// Project Hardware Driver layer. This is the only POU that accesses GVL_PressIO.
// It maps raw process-image symbols to semantic HALs and refreshes the Core
// topology publisher. It contains no sequence, mode, recipe or device behavior.
FUNCTION_BLOCK FB_PressIoDriver
VAR_OUTPUT
    // Raw N54 D2 operator buttons, republished so MAIN can drive Control On/Off
    // from hardware without becoming a second GVL_PressIO consumer.
    ControlOnButton  : BOOL;
    ControlOffButton : BOOL;
END_VAR
VAR
    _publisher : FB_IoTopologyPublisher;
    {attribute 'OPC.UA.DA' := '0'}
    _unit : REFERENCE TO FB_PressDemoUnit;
    _attached : BOOL;
    // Hardware Control-On adapter: reconstructs the safety-status mirrors from
    // the raw relay/sensor process image on a machine with a hardwired N54 D2
    // Control On circuit (no TwinSAFE controller). Status only; not a safety fn.
    _controlOn : FB_PressControlOnCircuit;
    // Reads the REAL EtherCAT slave states from the master and publishes each
    // node's live state — the fieldbus tree reflects hardware, not Control-On.
    _busHealth : FB_EcBusHealth;
END_VAR

;

METHOD Setup : BOOL
VAR_INPUT
    UnitRef : REFERENCE TO FB_PressDemoUnit;
END_VAR
VAR
    // Left all-zero: FB_EcBusHealth auto-detects the EtherCAT master's AmsNetId,
    // so the project needs no fieldbus address and no XAE link. Assign a value
    // here only for a non-standard master (remote, or several on one PC).
    ecMasterNetId : T_AmsNetIdArr;
END_VAR
_unit REF= UnitRef;
_attached := _publisher.Setup(DataRef := GVL_PressFieldbus.Topology, ResetData := FALSE)
    AND __ISVALIDREF(_unit);
// Map the press topology to the EtherCAT master's slaves. The catalog defines
// node 1 = CX2030 master and nodes 2..6 = the five devices in the project tree
// (EK1200 coupler, EL1809, EL2809, EL6001, EL9011).
//
// Only THREE of those are slaves the master enumerates: the EK1200 coupler and
// the EL9011 end cap carry the bus but have no EtherCAT slave controller on the
// process-data ring, so they never appear in FB_EcGetAllSlaveStates. Declaring
// SlaveCount := 5 made the master's slave i land on catalog node i, shifting
// every state onto its neighbour: the EL6001's OP was published onto the
// EL2809, and the EL6001 itself read OFFLINE while it was perfectly healthy.
// State the mapping instead of assuming it.
_busHealth.Setup(Publisher := _publisher, MasterNetIdArr := ecMasterNetId,
    FirstSlaveNode := 3, SlaveCount := 3, MasterNodeIndex := 1);
_busHealth.M_MapSlaveNode(SlaveIndex := 1, NodeIndex := 3);   // EL1809
_busHealth.M_MapSlaveNode(SlaveIndex := 2, NodeIndex := 4);   // EL2809
_busHealth.M_MapSlaveNode(SlaveIndex := 3, NodeIndex := 5);   // EL6001
_busHealth.M_MapPassiveNode(NodeIndex := 2);                  // EK1200 coupler
_busHealth.M_MapPassiveNode(NodeIndex := 6);                  // EL9011 end cap
Setup := _attached;
END_METHOD

METHOD M_ReadInputs
VAR_IN_OUT
    PressHal : ST_CylinderHal;
    DoorHal : ST_CylinderHal;
    SlideHal : ST_CylinderHal;
    TwoHandHal : ST_TwoHandHal;
    PowerHal : ST_PowerGroupHal;
    PartPresentHal : ST_DigitalInputHal;
    AirPressureHal : ST_AirPressureHal;
    RawEStopHealthy : BOOL;
    SafeEStopOk : BOOL;
    SafeGuardClosed : BOOL;
    SafeTwoHandActive : BOOL;
    SafePneumaticPermit : BOOL;
    SafetyFieldbusHealthy : BOOL;
    StandardIoHealthy : BOOL;
END_VAR
VAR
    // EtherCAT process-image validity, DETECTED from the fieldbus master by the
    // library (FB_EcBusHealth) — the project no longer declares/links a RealBusOk.
    busOk : BOOL;
END_VAR
busOk := _busHealth.M_BusOk();
// Physical feeder retracted = logical slide inside; extended = outside.
SlideHal.ExtendedFb := GVL_PressIO._101B301A;
SlideHal.RetractedFb := GVL_PressIO._101B301B;
DoorHal.ExtendedFb := GVL_PressIO._101B201A;
DoorHal.RetractedFb := GVL_PressIO._101B201B;
PressHal.ExtendedFb := GVL_PressIO._101B202A;
PressHal.RetractedFb := GVL_PressIO._101B202B;
TwoHandHal.RightPressed := GVL_PressIO._101S101;
TwoHandHal.LeftPressed := GVL_PressIO._101S102;
PartPresentHal.Value := GVL_PressIO._101B601;
AirPressureHal.LowPressure := GVL_PressIO._000MB085A_2;
AirPressureHal.OperatingPressure := GVL_PressIO._000MB085A_4;
PowerHal.PowerFeedback := GVL_PressIO._000K911_Y32;
// This machine's safety is a hardwired N54 D2 Control On relay chain, not a
// TwinSAFE controller, so the GVL_PressSafety AT %I* aliases are never written.
// Reconstruct the read-only safety-status mirrors from the raw relay/sensor
// process image via the Control-On adapter. The relay chain remains the safety
// authority; these values drive HMI/interlock display only.
_controlOn.M_Evaluate(
    // POLARITY: =000+S1-K910A:14 is "Emergency Switch 1 PRESSED" (N54 D2), and on
    // THIS machine the contact is CONFIRMED NORMALLY OPEN - not pressed reads
    // FALSE, pressed reads TRUE - so inverting it yields the "healthy" mirror
    // this adapter publishes. Read un-inverted, a healthy machine reported
    // E-stop-unhealthy and control power was withheld (POWER_ENABLE_WITHHELD)
    // even with the relay chain demonstrably closed.
    //
    // DEMO WIRING ONLY - NOT FAIL-SAFE. A normally-open E-stop contact cannot
    // distinguish "not pressed" from a broken wire, a pulled terminal or a dead
    // input card: all read FALSE, and this mirror would then report HEALTHY.
    // ISO 13850 / EN 60204-1 require a normally-CLOSED contact so that any break
    // forces the stop. A production machine must rewire to NC and drop this
    // inversion. This mirror is diagnostic only - the hardwired relay chain
    // remains the safety authority (Core Sec.9), which is what keeps the
    // non-fail-safe wiring tolerable on a demo rig and nowhere else.
    EStopHealthyMirror := NOT GVL_PressIO._000K910A,
    DoorClosed := GVL_PressIO._101B201A,
    LeftButton := GVL_PressIO._101S102,
    RightButton := GVL_PressIO._101S101,
    ControlOnFeedback := GVL_PressIO._000K911_Y32,
    BusOk := busOk,
    ControlOnButton := GVL_PressIO._000BS901,
    ControlOffButton := GVL_PressIO._000BS902,
    AirPressureOk := GVL_PressIO._000MB085A_4 AND NOT GVL_PressIO._000MB085A_2);
RawEStopHealthy := _controlOn.RawEStopHealthy;
SafeEStopOk := _controlOn.SafeEStopOk;
SafeGuardClosed := _controlOn.SafeGuardClosed;
SafeTwoHandActive := _controlOn.SafeTwoHandActive;
SafePneumaticPermit := _controlOn.SafePneumaticPermit;
SafetyFieldbusHealthy := _controlOn.SafetyFieldbusHealthy;
StandardIoHealthy := _controlOn.StandardIoHealthy;
PartPresentHal.Quality := StandardIoHealthy;
AirPressureHal.Quality := StandardIoHealthy;
ControlOnButton := GVL_PressIO._000BS901;
ControlOffButton := GVL_PressIO._000BS902;
END_METHOD

// Also withdraws every held §10.5.1 force: under USE_SIMULATION no physical
// output is driven at all, so a set-point armed earlier must not survive here
// and reappear the moment a real write path runs (§10.5.1 rule 3).
METHOD M_ClearOutputs
_publisher.M_ApplyForces(Enabled := FALSE);
GVL_PressIO._101K301A := FALSE; GVL_PressIO._101K301B := FALSE;
GVL_PressIO._101K201A := FALSE; GVL_PressIO._101K201B := FALSE;
GVL_PressIO._101K202A := FALSE; GVL_PressIO._101K202B := FALSE;
GVL_PressIO._101P101 := FALSE; GVL_PressIO._101P102 := FALSE;
GVL_PressIO._000K951_A1 := FALSE; GVL_PressIO._000K911_A1 := FALSE;
END_METHOD

METHOD M_WriteOutputs
VAR_INPUT
    PressHal : ST_CylinderHal;
    DoorHal : ST_CylinderHal;
    SlideHal : ST_CylinderHal;
    PowerHal : ST_PowerGroupHal;
    LampsOn : BOOL;
    ControlCircuitMappingConfirmed : BOOL;
    // Core §10.5.1 rule 3 - FB_UnitBase.M_ForcePermitted() of the owning Unit.
    // The SAME predicate its ForceChannel accepted the request with, so a force
    // can never be accepted under conditions in which it would not be applied,
    // and leaving idle MANUAL withdraws every held set-point on that scan.
    ForcePermitted : BOOL;
END_VAR
// One call decides whether held set-points apply this scan, and withdraws them
// all on the falling edge. It runs BEFORE the writes below, so the very scan
// the Unit leaves idle MANUAL is already driven by application logic again.
_publisher.M_ApplyForces(Enabled := ForcePermitted);
// M_EffectiveBool returns the value, so each line still reads as the plain
// assignment it was: the application value, or the held force set-point while
// forcing is permitted and this channel is forced.
GVL_PressIO._101K301A := _publisher.M_EffectiveBool(NodeIndex := 4, ChannelIndex := 1, Value := SlideHal.ExtendOut);
GVL_PressIO._101K301B := _publisher.M_EffectiveBool(NodeIndex := 4, ChannelIndex := 2, Value := SlideHal.RetractOut);
GVL_PressIO._101K201A := _publisher.M_EffectiveBool(NodeIndex := 4, ChannelIndex := 3, Value := DoorHal.ExtendOut);
GVL_PressIO._101K201B := _publisher.M_EffectiveBool(NodeIndex := 4, ChannelIndex := 4, Value := DoorHal.RetractOut);
GVL_PressIO._101K202A := _publisher.M_EffectiveBool(NodeIndex := 4, ChannelIndex := 5, Value := PressHal.ExtendOut);
GVL_PressIO._101K202B := _publisher.M_EffectiveBool(NodeIndex := 4, ChannelIndex := 6, Value := PressHal.RetractOut);
GVL_PressIO._101P101 := _publisher.M_EffectiveBool(NodeIndex := 4, ChannelIndex := 7, Value := LampsOn);
GVL_PressIO._101P102 := _publisher.M_EffectiveBool(NodeIndex := 4, ChannelIndex := 8, Value := LampsOn);
// Ch9/Ch10 (_000K951_A1 / _000K911_A1) are never routed through the force
// path: they drive the hardwired N54 D2 Control On relay chain and the
// catalog never marks them forceable (§10.5.1 rule 4).
IF ControlCircuitMappingConfirmed THEN
    // N54 D2: these are DIFFERENT signals. SwitchControlOn is the momentary
    // button coil (2 s pulse); EnableControlOn is the bus/air permissive that
    // must be TRUE whenever the machine is healthy. Driving both from one power
    // request was why the control circuit could never energize.
    GVL_PressIO._000K951_A1 := _controlOn.SwitchControlOn;
    GVL_PressIO._000K911_A1 := _controlOn.EnableControlOn;
ELSE
    GVL_PressIO._000K951_A1 := FALSE;
    GVL_PressIO._000K911_A1 := FALSE;
END_IF
END_METHOD

// The EtherCAT adapter this driver owns, handed once to the health probe by the
// composition root (§8.12/§10.5): one master, sampled once, read by both.
METHOD M_BusHealth : POINTER TO FB_EcBusHealth
M_BusHealth := ADR(_busHealth);
END_METHOD

// Node state now comes from the REAL EtherCAT master (FB_EcBusHealth), NOT from
// the Control-On / StandardIoHealthy verdict — the HMI fieldbus tree mirrors
// the actual bus (as XAE shows it). StandardIoHealthy is no longer an input.
METHOD M_RefreshFieldbus
VAR_INPUT
    // §10.5.1: the bus picture is a diagnostic surface, so the master is only
    // scanned while a consumer is actually reading it (the HMI fieldbus view is
    // open). Pass FALSE to park the scan; published states are then held, not
    // invalidated. One scan always runs after Setup so M_BusOk() has real data.
    BusViewActive : BOOL;
END_VAR
VAR
    D : ST_Diagnostic;
END_VAR
IF _attached THEN
    _busHealth.M_RequestScan(Active := BusViewActive);
    _busHealth.M_Refresh();  // publishes each node's real INIT/PREOP/SAFEOP/OP/FAULT
    _publisher.M_SetDigitalValue(NodeIndex := 3, ChannelIndex := 1, Value := GVL_PressIO._101B301A);
    _publisher.M_SetDigitalValue(NodeIndex := 3, ChannelIndex := 2, Value := GVL_PressIO._101B301B);
    _publisher.M_SetDigitalValue(NodeIndex := 3, ChannelIndex := 3, Value := GVL_PressIO._101B201A);
    _publisher.M_SetDigitalValue(NodeIndex := 3, ChannelIndex := 4, Value := GVL_PressIO._101B201B);
    _publisher.M_SetDigitalValue(NodeIndex := 3, ChannelIndex := 5, Value := GVL_PressIO._101B202A);
    _publisher.M_SetDigitalValue(NodeIndex := 3, ChannelIndex := 6, Value := GVL_PressIO._101B202B);
    _publisher.M_SetDigitalValue(NodeIndex := 3, ChannelIndex := 7, Value := GVL_PressIO._101S101);
    _publisher.M_SetDigitalValue(NodeIndex := 3, ChannelIndex := 8, Value := GVL_PressIO._101S102);
    _publisher.M_SetDigitalValue(NodeIndex := 3, ChannelIndex := 9, Value := GVL_PressIO._000MB085A_2);
    _publisher.M_SetDigitalValue(NodeIndex := 3, ChannelIndex := 10, Value := GVL_PressIO._000MB085A_4);
    _publisher.M_SetDigitalValue(NodeIndex := 3, ChannelIndex := 11, Value := GVL_PressIO._101B601);
    _publisher.M_SetDigitalValue(NodeIndex := 3, ChannelIndex := 12, Value := GVL_PressIO._000K911_Y32);
    _publisher.M_SetDigitalValue(NodeIndex := 3, ChannelIndex := 13, Value := GVL_PressIO._000K910A);
    _publisher.M_SetDigitalValue(NodeIndex := 4, ChannelIndex := 1, Value := GVL_PressIO._101K301A);
    _publisher.M_SetDigitalValue(NodeIndex := 4, ChannelIndex := 2, Value := GVL_PressIO._101K301B);
    _publisher.M_SetDigitalValue(NodeIndex := 4, ChannelIndex := 3, Value := GVL_PressIO._101K201A);
    _publisher.M_SetDigitalValue(NodeIndex := 4, ChannelIndex := 4, Value := GVL_PressIO._101K201B);
    _publisher.M_SetDigitalValue(NodeIndex := 4, ChannelIndex := 5, Value := GVL_PressIO._101K202A);
    _publisher.M_SetDigitalValue(NodeIndex := 4, ChannelIndex := 6, Value := GVL_PressIO._101K202B);
    _publisher.M_SetDigitalValue(NodeIndex := 4, ChannelIndex := 7, Value := GVL_PressIO._101P101);
    _publisher.M_SetDigitalValue(NodeIndex := 4, ChannelIndex := 8, Value := GVL_PressIO._101P102);
    _publisher.M_SetDigitalValue(NodeIndex := 4, ChannelIndex := 9, Value := GVL_PressIO._000K951_A1);
    _publisher.M_SetDigitalValue(NodeIndex := 4, ChannelIndex := 10, Value := GVL_PressIO._000K911_A1);
    _publisher.M_BeginDiagnosticRefresh();
    D := _unit.PressRam.Status.Diagnostic;
    _M_ApplyCylinderDiagnostic(Diagnostic := D,
        ExtendedTag := _unit.PressRam.OutImm.ExtendedSensorTag,
        RetractedTag := _unit.PressRam.OutImm.RetractedSensorTag);
    D := _unit.Door.Status.Diagnostic;
    _M_ApplyCylinderDiagnostic(Diagnostic := D,
        ExtendedTag := _unit.Door.OutImm.ExtendedSensorTag,
        RetractedTag := _unit.Door.OutImm.RetractedSensorTag);
    D := _unit.PartSlide.Status.Diagnostic;
    _M_ApplyCylinderDiagnostic(Diagnostic := D,
        ExtendedTag := _unit.PartSlide.OutImm.ExtendedSensorTag,
        RetractedTag := _unit.PartSlide.OutImm.RetractedSensorTag);
    D := _unit.AirPressureMonitor.Status.Diagnostic;
    _publisher.M_ApplyDiagnostic(Diagnostic := D);
    IF TO_DINT(D.ReasonCode) = PL_ModuleReasons.AIR_SWITCH_CONFLICT THEN
        _publisher.M_ApplyDiagnosticToTag(Diagnostic := D,
            Tag := _unit.AirPressureMonitor.OutImm.LowSensorTag);
        _publisher.M_ApplyDiagnosticToTag(Diagnostic := D,
            Tag := _unit.AirPressureMonitor.OutImm.OperatingSensorTag);
    ELSE
        ;
    END_IF
    // §10.5.1 — the RS232 terminal's process image, published like any other
    // channel so a dead serial link is visible on the bus page instead of invisible.
    _publisher.M_SetAnalogValue(NodeIndex := 5, ChannelIndex := 1, Value := USINT_TO_REAL(GVL_PressIO._000K010D1_Status));
    _publisher.M_SetAnalogValue(NodeIndex := 5, ChannelIndex := 2, Value := USINT_TO_REAL(GVL_PressIO._000K010D1_DataIn0));
    _publisher.M_SetAnalogValue(NodeIndex := 5, ChannelIndex := 3, Value := USINT_TO_REAL(GVL_PressIO._000K010D1_DataIn1));
    _publisher.M_SetAnalogValue(NodeIndex := 5, ChannelIndex := 4, Value := USINT_TO_REAL(GVL_PressIO._000K010D1_DataIn2));
    _publisher.M_SetAnalogValue(NodeIndex := 5, ChannelIndex := 5, Value := USINT_TO_REAL(GVL_PressIO._000K010D1_Ctrl));
    _publisher.M_SetAnalogValue(NodeIndex := 5, ChannelIndex := 6, Value := USINT_TO_REAL(GVL_PressIO._000K010D1_DataOut0));
    _publisher.M_SetAnalogValue(NodeIndex := 5, ChannelIndex := 7, Value := USINT_TO_REAL(GVL_PressIO._000K010D1_DataOut1));
    _publisher.M_SetAnalogValue(NodeIndex := 5, ChannelIndex := 8, Value := USINT_TO_REAL(GVL_PressIO._000K010D1_DataOut2));
    _publisher.M_ApplyDiagnostic(Diagnostic := _unit.Status.Diagnostic);
ELSE
    ;
END_IF
END_METHOD

METHOD PRIVATE _M_ApplyCylinderDiagnostic
VAR_INPUT
    Diagnostic : ST_Diagnostic;
    ExtendedTag : STRING(80);
    RetractedTag : STRING(80);
END_VAR
_publisher.M_ApplyDiagnostic(Diagnostic := Diagnostic);
IF TO_DINT(Diagnostic.ReasonCode) = PL_ModuleReasons.CYL_BOTH_SENSORS THEN
    _publisher.M_ApplyDiagnosticToTag(Diagnostic := Diagnostic, Tag := ExtendedTag);
    _publisher.M_ApplyDiagnosticToTag(Diagnostic := Diagnostic, Tag := RetractedTag);
ELSE
    ;
END_IF
END_METHOD

END_FUNCTION_BLOCK

(* stored: Version 1.1.0.1, ProductVersion 3.1.4024.12
   POU FB_PressIoDriver: Id {bedb7de0-6ee7-499c-942c-a47bd1ba5582}, SpecialFunc None
   Method Setup: Id {3d2dc4cb-5c7c-441c-b71b-e76c6dc5e5ea}
   Method M_ReadInputs: Id {0808b97f-7dcc-44e8-9480-17a48c17ac6f}
   Method M_ClearOutputs: Id {f625a4c1-e10f-4e07-b91a-6885860994d0}
   Method M_WriteOutputs: Id {cc5ac6ba-fd45-445f-908c-0307380375bc}
   Method M_BusHealth: Id {f61f7ebd-dc5e-472b-8981-448a39505162}
   Method M_RefreshFieldbus: Id {69fbd59b-ae26-4b9d-9552-541f2a36a52b}
   Method _M_ApplyCylinderDiagnostic: Id {c5bd449b-e7c7-4d49-8755-d2386bdfef10} *)
